PROGRAM MAIN
VAR
END_VAR

LenzeServoDrive();

END_PROGRAM

(* stored: Version 1.1.0.1, ProductVersion 3.1.4024.12
   POU MAIN: Id {a2221aa7-ca8f-4b9b-a5e0-2ad25a564e89}, SpecialFunc None *)
